// TIA Portal V15.1 export
// export: Created 2024-06-21T08:41:21.2804281Z, ExportSetting WithDefaults, DisplayName Totally Integrated Automation Portal, DisplayVersion V15.1 Update 5, DisplayName TIA Portal Openness, DisplayVersion V15.1 Update 5, DisplayName SINAMICS Startdrive Advanced, DisplayVersion V15.1, DisplayName G130, G150, S120, S150, SINAMICS MV, S210, DisplayVersion V15.1, DisplayName G110M, G120, G120C, G120D, G120P, DisplayVersion V15.1, DisplayName STEP 7 Professional, DisplayVersion V15.1 Update 5, DisplayName STEP 7 Safety, DisplayVersion V15.1, DisplayName WinCC Professional, DisplayVersion V15.1 Update 5, DisplayName SIMATIC Visualization Architect, DisplayVersion V15.1
FUNCTION_BLOCK "LVIDSDeCouple"   // FB1208, SCL
{ S7_Optimized_Access := 'TRUE' }
VERSION : 0.1
// stored: AutoNumber false, IsIECCheckEnabled false, IsRetainMemResEnabled false, MemoryReserve 100, SetENOAutomatically False, UDAEnableTagReadback false
   VAR_INPUT
      C_SoftCouple { ExternalAccessible := 'False'; ExternalVisible := 'False'; ExternalWritable := 'False'} : Bool;   // If true, coupling between CarrierID and BodyID or Mixnumber, otherwise with TagID
      I_DataModeManEn { ExternalAccessible := 'False'; ExternalVisible := 'False'; ExternalWritable := 'False'} : Bool;   // Dat mode manual enabled
      I_TagID { ExternalAccessible := 'False'; ExternalVisible := 'False'; ExternalWritable := 'False'} : DWord;   // Received TagId to couple with Data / Tag ID (0 if not used)
      I_BodyID { ExternalAccessible := 'False'; ExternalVisible := 'False'; ExternalWritable := 'False'} : DWord;   // Bodynumber (0 if not used)
      I_CarrierID { ExternalAccessible := 'False'; ExternalVisible := 'False'; ExternalWritable := 'False'} : DWord;   // Carrier ID
      I_MixNbr { ExternalAccessible := 'False'; ExternalVisible := 'False'; ExternalWritable := 'False'} : DWord;   // Mixnumber (0 if not used)
      I_PopID { ExternalAccessible := 'False'; ExternalVisible := 'False'; ExternalWritable := 'False'} : UDInt;   // Spare Data / PopID (0 if not used)
      I_PopIDSuffix { ExternalAccessible := 'False'; ExternalVisible := 'False'; ExternalWritable := 'False'} : Char;   // PopID suffix (' ' if not used)
      I_PopType { ExternalAccessible := 'False'; ExternalVisible := 'False'; ExternalWritable := 'False'} : UDInt;   // Pop identifier
      I_Start { ExternalAccessible := 'False'; ExternalVisible := 'False'; ExternalWritable := 'False'} : Bool;   // Start command for coupling / Start command
   END_VAR
   VAR_OUTPUT
      O_DataModeAuto { ExternalAccessible := 'False'; ExternalVisible := 'False'; ExternalWritable := 'False'} : Bool;   // Couple or decouple in automatic mode / Data mode - Automatic
      O_DataModeMan { ExternalAccessible := 'False'; ExternalVisible := 'False'; ExternalWritable := 'False'} : Bool;   // Data mode - Manual
      O_Busy { ExternalAccessible := 'False'; ExternalVisible := 'False'; ExternalWritable := 'False'} : Bool;   // Coupling busy
      O_Status { ExternalAccessible := 'False'; ExternalVisible := 'False'; ExternalWritable := 'False'} : Int;   // Status / Status (< 0 : alarm)
      O_Alarm { ExternalAccessible := 'False'; ExternalVisible := 'False'; ExternalWritable := 'False'} : Bool;   // Alarm
      O_OK { ExternalAccessible := 'False'; ExternalVisible := 'False'; ExternalWritable := 'False'} : Bool;   // Coupling or decoupling done OK / Coupling OK
      O_NOK { ExternalAccessible := 'False'; ExternalVisible := 'False'; ExternalWritable := 'False'} : Bool;   // Coupling or decoupling done NOK / Coupling NOK
   END_VAR
   VAR_IN_OUT
      IO_VIDS : "VIDS";   // VIDS internal record
      IO_VEMData : "VEMData";   // VEM data (From master)
      IO_Alarm : "Alarm";   // Alarm
      H_DeCouple : "H_LVIDSDeCouple";
      H_HMI : "H_HMI";
   END_VAR
   VAR
      DataModeAuto { ExternalAccessible := 'False'; ExternalVisible := 'False'; ExternalWritable := 'False'} : Bool;   // Couple or decouple in automode
      DataModeAutoPls { ExternalAccessible := 'False'; ExternalVisible := 'False'; ExternalWritable := 'False'} : Bool;
      DataModeMan { ExternalAccessible := 'False'; ExternalVisible := 'False'; ExternalWritable := 'False'} : Bool;
      DataModeManPls { ExternalAccessible := 'False'; ExternalVisible := 'False'; ExternalWritable := 'False'} : Bool;
      DataModeEdit { ExternalAccessible := 'False'; ExternalVisible := 'False'; ExternalWritable := 'False'} : Bool;
      DataModeMem { ExternalAccessible := 'False'; ExternalVisible := 'False'; ExternalWritable := 'False'} : Int;
      DataModeChanged { ExternalAccessible := 'False'; ExternalVisible := 'False'; ExternalWritable := 'False'} : Bool;
      DeCoupleBeginReqPlsAuto { ExternalAccessible := 'False'; ExternalVisible := 'False'; ExternalWritable := 'False'} : Bool;
      DeCoupleBeginReqPlsMan { ExternalAccessible := 'False'; ExternalVisible := 'False'; ExternalWritable := 'False'} : Bool;
      StartPls { ExternalAccessible := 'False'; ExternalVisible := 'False'; ExternalWritable := 'False'} : Bool;
      BeginReqAuto { ExternalAccessible := 'False'; ExternalVisible := 'False'; ExternalWritable := 'False'} : Bool;
      Busy { ExternalAccessible := 'False'; ExternalVisible := 'False'; ExternalWritable := 'False'} : Bool;
      BeginReqMan { ExternalAccessible := 'False'; ExternalVisible := 'False'; ExternalWritable := 'False'} : Bool;
      CarrierID { ExternalAccessible := 'False'; ExternalVisible := 'False'; ExternalWritable := 'False'} : DWord;
      CarrierIDValid { ExternalAccessible := 'False'; ExternalVisible := 'False'; ExternalWritable := 'False'} : Bool;
   END_VAR
   VAR DB_SPECIFIC
      CarrierIDMem { ExternalAccessible := 'False'; ExternalVisible := 'False'; ExternalWritable := 'False'} : DWord;   // Memory of CarrierID at begin request
   END_VAR
   VAR
      Identification { ExternalAccessible := 'False'; ExternalVisible := 'False'; ExternalWritable := 'False'} : DWord;
      IdentificationValid { ExternalAccessible := 'False'; ExternalVisible := 'False'; ExternalWritable := 'False'} : Bool;
      IdentificationMem { ExternalAccessible := 'False'; ExternalVisible := 'False'; ExternalWritable := 'False'} : DWord;
      BodyNbr { ExternalAccessible := 'False'; ExternalVisible := 'False'; ExternalWritable := 'False'} : DWord;
      BodyNbrValid { ExternalAccessible := 'False'; ExternalVisible := 'False'; ExternalWritable := 'False'} : Bool;
      BodyIDMem { ExternalAccessible := 'False'; ExternalVisible := 'False'; ExternalWritable := 'False'} : DWord;
      MixNbr { ExternalAccessible := 'False'; ExternalVisible := 'False'; ExternalWritable := 'False'} : DWord;
      MixNbrValid { ExternalAccessible := 'False'; ExternalVisible := 'False'; ExternalWritable := 'False'} : Bool;
      MixNbrMem { ExternalAccessible := 'False'; ExternalVisible := 'False'; ExternalWritable := 'False'} : DWord;
      PopIDMem { ExternalAccessible := 'False'; ExternalVisible := 'False'; ExternalWritable := 'False'} : DWord;
      PopIDSuffixMem { ExternalAccessible := 'False'; ExternalVisible := 'False'; ExternalWritable := 'False'} : Char;
      PopTypeMem { ExternalAccessible := 'False'; ExternalVisible := 'False'; ExternalWritable := 'False'} : DWord;
      DataValid { ExternalAccessible := 'False'; ExternalVisible := 'False'; ExternalWritable := 'False'} : Bool;
      InputDataValidAuto { ExternalAccessible := 'False'; ExternalVisible := 'False'; ExternalWritable := 'False'} : Bool;
      InputDataValidMan { ExternalAccessible := 'False'; ExternalVisible := 'False'; ExternalWritable := 'False'} : Bool;
      DataNotValid { ExternalAccessible := 'False'; ExternalVisible := 'False'; ExternalWritable := 'False'} : Bool;
   END_VAR
   VAR DB_SPECIFIC
      BeginPlsModeAuto { ExternalAccessible := 'False'; ExternalVisible := 'False'; ExternalWritable := 'False'} : Bool;   // Pulse of begin in auto mode
      BeginPlsModeManTagId { ExternalAccessible := 'False'; ExternalVisible := 'False'; ExternalWritable := 'False'} : Bool;   // Pulse of begin in manual mode
      BeginReqPls { ExternalAccessible := 'False'; ExternalVisible := 'False'; ExternalWritable := 'False'} : Bool;   // Pulse of begin request
      TagIdModeManMem { ExternalAccessible := 'False'; ExternalVisible := 'False'; ExternalWritable := 'False'} : DWord;   // Memorised TagId in manual mode
      Alarm { ExternalAccessible := 'False'; ExternalVisible := 'False'; ExternalWritable := 'False'} : Bool;   // Alarm
      ChangedRcvDataAlarm { ExternalAccessible := 'False'; ExternalVisible := 'False'; ExternalWritable := 'False'} : Bool;   // Alarm received data has chnged after request
      CoupleAlarm { ExternalAccessible := 'False'; ExternalVisible := 'False'; ExternalWritable := 'False'} : Bool;   // Alarm couple or decouple NOK
      Status { ExternalAccessible := 'False'; ExternalVisible := 'False'; ExternalWritable := 'False'} : Int;   // Status
   END_VAR
   VAR
      btnDataModeAutoColour { ExternalAccessible := 'False'; ExternalVisible := 'False'; ExternalWritable := 'False'} : Word;
      btnDataModeManColour { ExternalAccessible := 'False'; ExternalVisible := 'False'; ExternalWritable := 'False'} : Word;
      btnDeCoupleVisible { ExternalAccessible := 'False'; ExternalVisible := 'False'; ExternalWritable := 'False'} : Word;
      btnDeCoupleEnable { ExternalAccessible := 'False'; ExternalVisible := 'False'; ExternalWritable := 'False'} : Word;
      btnDeCouplePls { ExternalAccessible := 'False'; ExternalVisible := 'False'; ExternalWritable := 'False'} : Bool;
      btnEditVisible { ExternalAccessible := 'False'; ExternalVisible := 'False'; ExternalWritable := 'False'} : Word;
      btnEditEnable { ExternalAccessible := 'False'; ExternalVisible := 'False'; ExternalWritable := 'False'} : Word;
      msgVEMDataBodyVisible { ExternalAccessible := 'False'; ExternalVisible := 'False'; ExternalWritable := 'False'} : Word;
      msgVEMDataCarrierVisible { ExternalAccessible := 'False'; ExternalVisible := 'False'; ExternalWritable := 'False'} : Word;
      msgDataValidVisible { ExternalAccessible := 'False'; ExternalVisible := 'False'; ExternalWritable := 'False'} : Word;   // HMI - Couple/Decouple OK
      msgDataNotValidVisible { ExternalAccessible := 'False'; ExternalVisible := 'False'; ExternalWritable := 'False'} : Word;   // HMI - Couple/Decouple OK
      msgPartPresVisible { ExternalAccessible := 'False'; ExternalVisible := 'False'; ExternalWritable := 'False'} : Word;
      txtCarrierIDDeCoupleVisible { ExternalAccessible := 'False'; ExternalVisible := 'False'; ExternalWritable := 'False'} : Word;
      txtCarrierIDDeCoupleEnable { ExternalAccessible := 'False'; ExternalVisible := 'False'; ExternalWritable := 'False'} : Word;
      txtCarrierIDDeCoupleColour { ExternalAccessible := 'False'; ExternalVisible := 'False'; ExternalWritable := 'False'} : Word;
      txtCarrierIDDeCoupleValid { ExternalAccessible := 'False'; ExternalVisible := 'False'; ExternalWritable := 'False'} : Bool;
      txtIdentificationDeCoupleVisible { ExternalAccessible := 'False'; ExternalVisible := 'False'; ExternalWritable := 'False'} : Word;
      txtIdentificationDeCoupleEnable { ExternalAccessible := 'False'; ExternalVisible := 'False'; ExternalWritable := 'False'} : Word;
      txtIdentificationDeCoupleColour { ExternalAccessible := 'False'; ExternalVisible := 'False'; ExternalWritable := 'False'} : Word;
      txtIdentificationDeCoupleValid { ExternalAccessible := 'False'; ExternalVisible := 'False'; ExternalWritable := 'False'} : Bool;
      txtMixNbrDeCoupleVisible { ExternalAccessible := 'False'; ExternalVisible := 'False'; ExternalWritable := 'False'} : Word;
      txtMixNbrDeCoupleEnable { ExternalAccessible := 'False'; ExternalVisible := 'False'; ExternalWritable := 'False'} : Word;
      txtMixNbrDeCoupleColour { ExternalAccessible := 'False'; ExternalVisible := 'False'; ExternalWritable := 'False'} : Word;
      txtMixNbrDeCoupleValid { ExternalAccessible := 'False'; ExternalVisible := 'False'; ExternalWritable := 'False'} : Bool;
      txtBodyIDDeCoupleVisible { ExternalAccessible := 'False'; ExternalVisible := 'False'; ExternalWritable := 'False'} : Word;
      txtBodyIDDeCoupleEnable { ExternalAccessible := 'False'; ExternalVisible := 'False'; ExternalWritable := 'False'} : Word;
      txtBodyIDDeCoupleColour { ExternalAccessible := 'False'; ExternalVisible := 'False'; ExternalWritable := 'False'} : Word;
      txtBodyIDDeCoupleValid { ExternalAccessible := 'False'; ExternalVisible := 'False'; ExternalWritable := 'False'} : Bool;
      txtPopIDDeCoupleVisible { ExternalAccessible := 'False'; ExternalVisible := 'False'; ExternalWritable := 'False'} : Word;
      txtPopIDDeCoupleEnable { ExternalAccessible := 'False'; ExternalVisible := 'False'; ExternalWritable := 'False'} : Word;
      txtPopIDDeCoupleColour { ExternalAccessible := 'False'; ExternalVisible := 'False'; ExternalWritable := 'False'} : Word;
      txtPopIDDeCoupleValid { ExternalAccessible := 'False'; ExternalVisible := 'False'; ExternalWritable := 'False'} : Bool;
      txtPopIDSuffixDeCoupleVisible { ExternalAccessible := 'False'; ExternalVisible := 'False'; ExternalWritable := 'False'} : Word;
      txtPopIDSuffixDeCoupleEnable { ExternalAccessible := 'False'; ExternalVisible := 'False'; ExternalWritable := 'False'} : Word;
      txtPopIDSuffixDeCoupleColour { ExternalAccessible := 'False'; ExternalVisible := 'False'; ExternalWritable := 'False'} : Word;
      txtPopTypeDeCoupleVisible { ExternalAccessible := 'False'; ExternalVisible := 'False'; ExternalWritable := 'False'} : Word;
      txtPopTypeDeCoupleEnable { ExternalAccessible := 'False'; ExternalVisible := 'False'; ExternalWritable := 'False'} : Word;
      txtPopTypeDeCoupleColour { ExternalAccessible := 'False'; ExternalVisible := 'False'; ExternalWritable := 'False'} : Word;
      IconColour { ExternalAccessible := 'False'; ExternalVisible := 'False'; ExternalWritable := 'False'} : Word;
      DeCoupleOK { ExternalAccessible := 'False'; ExternalVisible := 'False'; ExternalWritable := 'False'} : Bool;
      DeCoupleNOK { ExternalAccessible := 'False'; ExternalVisible := 'False'; ExternalWritable := 'False'} : Bool;
      _DataModeManForcedPls { ExternalAccessible := 'False'; ExternalVisible := 'False'; ExternalWritable := 'False'; S7_SetPoint := 'True'} : R_TRIG;
      _DataModeAutoPls { ExternalAccessible := 'False'; ExternalVisible := 'False'; ExternalWritable := 'False'; S7_SetPoint := 'True'} : R_TRIG;
      _DeCoupleStartPls { ExternalAccessible := 'False'; ExternalVisible := 'False'; ExternalWritable := 'False'; S7_SetPoint := 'True'} : R_TRIG;
      _DataModeChangedPls { ExternalAccessible := 'False'; ExternalVisible := 'False'; ExternalWritable := 'False'; S7_SetPoint := 'True'} : R_TRIG;
      _btnDeCouplePls { ExternalAccessible := 'False'; ExternalVisible := 'False'; ExternalWritable := 'False'; S7_SetPoint := 'True'} : R_TRIG;
   END_VAR
   VAR CONSTANT
      STATUS_OK : Int := 1;
      STATUS_COUPLE_REQ : Int := 107;
      STATUS_COUPLE_RUNNING : Int := 207;
      STATUS_DECOUPLE_REQ : Int := 108;
      STATUS_DECOUPLE_RUNNING : Int := 208;
      OFF : Word := 2#0000000000000000;
      ON : Word := 2#0000000000000001;
      VISIBLE : Word := 2#0000000000000001;
      ENABLE : Word := 2#0000000000000010;
      BG_COLOUR_GREY : Word := 2#0000000000000100;
      COLOUR_DEFAULT : Word := 2#0000000000000000;
      COLOUR_RED : Word := 2#0000000000010000;
      COLOUR_GREEN : Word := 2#0000000000100000;
      COLOUR_BLUE : Word := 2#0000000001000000;
      COLOUR_WHITE : Word := 2#0000000010000000;
      BG_COLOUR_BLUE_FLASH : Word := 2#0000000010000000;
      BG_COLOUR_LIGHTRED : Word := 2#0100000000000000;
      BG_COLOUR_YELLOW : Word := 2#1000000000000000;
      OK_BEGIN_DELAY_MAX : Time := T#10s;
      CMD_DECOUPLE : DWord := 2006;
   END_VAR
BEGIN
   (******************************************************************************)
   (* Data mode - Activation                                                     *)
   (******************************************************************************)

   //Automatic
   //Data mode selected  - No mode, select auto
   IF (#H_DeCouple.H_selDataMode < 1) OR (#H_DeCouple.H_selDataMode > 3) OR NOT #IO_VIDS.PartPres OR NOT #I_DataModeManEn THEN
       #H_DeCouple.H_selDataMode := 1;
   END_IF;

   //Data mode automatic - Activation
   #DataModeAuto := (#H_DeCouple.H_selDataMode = 1);

   //Data mode automatic - Create pulse upon selection 
   #_DataModeAutoPls(CLK:=#DataModeAuto,Q=>#DataModeAutoPls);

   //Data mode manual - Activation
   #DataModeMan := (#H_DeCouple.H_selDataMode = 2);

   //Data mode manual - Create pulse upon selection
   #_DataModeManForcedPls(CLK := #DataModeMan,Q => #DataModeManPls);

   //Data mode changed
   #_DataModeAutoPls(CLK := #H_DeCouple.H_selDataMode <> #DataModeMem,Q => #DataModeAutoPls);
   #DataModeMem:=#H_DeCouple.H_selDataMode;

   //Data mode edit - Activation
   IF #DataModeMan AND (#H_DeCouple.H_btnEdit = #ON) THEN
       #DataModeEdit := TRUE;
       //Copy VEM data to HMI
       #H_DeCouple.H_txtIdentification := #IO_VEMData.Identification;

   ELSIF #DataModeAuto THEN
       #DataModeEdit := FALSE;
   END_IF;


   IF #DataModeEdit THEN

       //Check valid
       #txtCarrierIDDeCoupleValid := #H_DeCouple.H_txtCarrierIDDeCouple > 0;
       #txtIdentificationDeCoupleValid := #H_DeCouple.H_txtIdentificationDeCouple > 0;
       #txtBodyIDDeCoupleValid :=#H_DeCouple.H_txtBodyIDDeCouple > 0;
       #txtMixNbrDeCoupleValid := #H_DeCouple.H_txtMixNbrDeCouple > 0;
       #txtPopIDDeCoupleValid := #H_DeCouple.H_txtPopIdDeCouple > 0;

       //Entry fields valid
       #InputDataValidMan := #txtCarrierIDDeCoupleValid AND (#txtIdentificationDeCoupleValid OR #txtBodyIDDeCoupleValid OR #txtMixNbrDeCoupleValid OR #txtPopIDDeCoupleValid);

   ELSE

       //Reset
       #InputDataValidMan := FALSE;

   END_IF;

   (******************************************************************************)
   (* Data mode automatic - Begin request                                        *)
   (******************************************************************************)

   //Start - Create pulse
   #_DeCoupleStartPls(CLK := #I_Start,
                    Q => #StartPls);

   #BeginReqAuto:=False;
   IF #DataModeAuto AND #StartPls AND #IO_VIDS.PartPres AND #I_CarrierID > 0  THEN

       //Memorize parameters
       #IdentificationMem := #I_TagID;
       #BodyIDMem := #I_BodyID;
       #CarrierIDMem := #I_CarrierID;
       #MixNbrMem := #I_MixNbr;
       #PopIDMem := #I_PopID;
       #PopIDSuffixMem := #I_PopIDSuffix;
       #PopTypeMem := #I_PopType;

       //Data mode automatic - Begin request
       #BeginReqAuto := True;

   END_IF;

   (******************************************************************************)
   (* Data mode manual - Begin request                                           *)
   (******************************************************************************)

   //Couple button - Create pulse 
   #_btnDeCouplePls(CLK:=#H_DeCouple.H_btnDecouple=#ON,
                  Q=>#btnDeCouplePls);

   #BeginReqMan := False;
   IF #DataModeEdit AND #btnDeCouplePls AND #IO_VIDS.PartPres THEN

       //Edit mode off
       #DataModeEdit := FALSE;

       //Memorize data
       #CarrierIDMem := #H_DeCouple.H_txtCarrierIDDeCouple;

       //Start with a clean sheet
       #IdentificationMem := 0;
       #BodyIDMem := 0;
       #MixNbrMem := 0;
       #PopIDMem := 0;
       #PopIDSuffixMem := ' ';
       #PopTypeMem := 0;

       //Memorize parameters
       IF #H_DeCouple.H_txtIdentificationDeCouple > 0 THEN
           #IdentificationMem := #H_DeCouple.H_txtIdentificationDeCouple;
       ELSIF #H_DeCouple.H_txtBodyIDDeCouple > 0 THEN
           #BodyIDMem := #H_DeCouple.H_txtBodyIDDeCouple;
       ELSIF #H_DeCouple.H_txtMixNbrDeCouple > 0 THEN
           #MixNbrMem := #H_DeCouple.H_txtMixNbrDeCouple;
       ELSIF #H_DeCouple.H_txtPopIdDeCouple > 0 OR #H_DeCouple.H_txtPopIdSuffixDeCouple <> ' ' OR #H_DeCouple.H_txtPopTypeDeCouple <> 0  THEN
           #PopIDMem := #H_DeCouple.H_txtPopIdDeCouple;
           #PopIDSuffixMem := #H_DeCouple.H_txtPopIdSuffixDeCouple;
           #PopTypeMem := #H_DeCouple.H_txtPopTypeDeCouple;
       END_IF;

       //Data mode manual - begin request
       #BeginReqMan := True;

   END_IF;

   (******************************************************************************)
   (* Begin request - Summary                                                    *)
   (******************************************************************************)

   #IO_VIDS.DeCouple.BeginReq := #BeginReqAuto OR #BeginReqMan;

   IF #IO_VIDS.DeCouple.BeginReq THEN
       #DeCoupleOK := False;
       #DeCoupleNOK := False;
   END_IF;

   (*******************************************************)
   (* Begin                                               *)
   (*******************************************************)

   IF #IO_VIDS.DeCouple.OkBegin THEN
       //Initialize parameters
       #IO_VIDS.VEMData.IdType := #IO_VIDS.IDType;
       #IO_VIDS.VEMData.FunctionCode := 255;
       #IO_VIDS.VEMData.Identification := #IdentificationMem;
       #IO_VIDS.VEMData.BodyID := #BodyIDMem;
       #IO_VIDS.VEMData.CarrierID := #CarrierIDMem;
       #IO_VIDS.VEMData.MixNumber := #MixNbrMem;
       #IO_VIDS.VEMData.PopID := #PopIDMem;
       #IO_VIDS.VEMData.PopIDSuffix := #PopIDSuffixMem;
       #IO_VIDS.VEMData.PopType := #PopTypeMem;
       #IO_VIDS.VEMData.CommandCode := #CMD_DECOUPLE;
       #Status := #IO_VIDS.DeCouple.Status;
   END_IF;

   #IO_VIDS.DeCouple.Begin := #IO_VIDS.DeCouple.OkBegin;

   (*******************************************************)
   (* Running                                             *)
   (*******************************************************)
   IF #IO_VIDS.DeCouple.Running THEN
       #Status := #IO_VIDS.DeCouple.Status;
   END_IF;

   #Busy := #IO_VIDS.DeCouple.Running;

   (*******************************************************)
   (* Finish                                              *)
   (*******************************************************)

   IF #IO_VIDS.DeCouple.Finished THEN

       //Update status
       #Status := #IO_VIDS.DeCouple.Status;

       //Status OK/NOK
       IF #Status = #STATUS_OK THEN
           #DeCoupleOK := True;
       ELSE
           #DeCoupleNOK := True;
           IF #DataModeMan THEN
               #DataModeEdit := TRUE;
           END_IF;
       END_IF;

   END_IF;

   (******************************************************************************)
   (* Alarm                                                                      *)
   (******************************************************************************)

   #Alarm := (#Status < 0);

   "LAlarmSummary"(I_AlarmA := "FALSE",
                   I_AlarmB := "FALSE",
                   I_AlarmC := #Alarm,
                   I_AlarmD := "FALSE",
                   I_AlarmABCondition := "FALSE",
                   IO_Alarm := #IO_Alarm,
                   C_UpperLevelHW := "FALSE",
                   C_UpperLevelSafety := "FALSE",
                   C_Safety := "FALSE",
                   C_Mechanic := "FALSE",
                   C_Transport := "FALSE",
                   C_Feature1 := "FALSE",
                   C_Feature2 := "FALSE",
                   C_Feature3 := "FALSE");


   (*******************************************************)
   (* Reset                                               *)
   (*******************************************************)

   IF NOT #IO_VIDS.PartPres THEN
       #DeCoupleOK := False;
       #DeCoupleNOK := False;
       #H_DeCouple.H_txtIdentification := 0;
       #H_DeCouple.H_txtBodyID := 0;
       #H_DeCouple.H_txtCarrierID := 0;
       #H_DeCouple.H_txtMixNbr := 0;
       #H_DeCouple.H_txtPopId := 0;
       #H_DeCouple.H_txtPopIdSuffix := ' ';
       #H_DeCouple.H_txtPopType := 0;
       #Status := 0;
   END_IF;

   (*******************************************************)
   (* Outputs                                             *)
   (*******************************************************)

   #O_DataModeAuto := #DataModeAuto;
   #O_DataModeMan := #DataModeMan;
   #O_OK := #DeCoupleOK;
   #O_NOK := #DeCoupleNOK;

   #O_Busy := #Busy;
   #O_Status := #Status;
   #O_Alarm := #Status < 0;

   (*******************************************************)
   (* HMI - Reset buttons                                 *)
   (*******************************************************)

   #H_DeCouple.H_btnEdit := #OFF;
   #H_DeCouple.H_btnDecouple := #OFF;
   #H_DeCouple.H_btnDecouple := #OFF;

   (*******************************************************)
   (* HMI - Update text fields                            *)
   (*******************************************************)

   IF #IO_VIDS.VEMDataValid THEN
       #H_DeCouple.H_txtCarrierIDDeCouple := #IO_VEMData.CarrierID;
       #H_DeCouple.H_txtIdentificationDeCouple := #IO_VEMData.Identification;
       #H_DeCouple.H_txtBodyIDDeCouple := #IO_VEMData.BodyID;
       #H_DeCouple.H_txtMixNbrDeCouple := #IO_VEMData.MixNumber;
       #H_DeCouple.H_txtPopId := #IO_VEMData.PopID;
       #H_DeCouple.H_txtPopIdSuffix := #IO_VEMData.PopIDSuffix;
       #H_DeCouple.H_txtPopType := #IO_VEMData.PopType;
   ELSE
       #H_DeCouple.H_txtCarrierID := 0;
       #H_DeCouple.H_txtIdentification := 0;
       #H_DeCouple.H_txtBodyID := 0;
       #H_DeCouple.H_txtMixNbr := 0;
       #H_DeCouple.H_txtPopId := 0;
       #H_DeCouple.H_txtPopIdSuffix := ' ';
       #H_DeCouple.H_txtPopType := 0;
   END_IF;

   (*******************************************************)
   (* HMI - Input fields                                  *)
   (*******************************************************)

   //Visible
   #txtIdentificationDeCoupleVisible := #OFF;
   #txtBodyIDDeCoupleVisible := #OFF;
   #txtCarrierIDDeCoupleVisible := #OFF;
   #txtMixNbrDeCoupleVisible := #OFF;
   #txtPopIDDeCoupleVisible := #OFF;
   #txtPopIDSuffixDeCoupleVisible := #OFF;
   #txtPopTypeDeCoupleVisible := #OFF;

   IF #DataModeMan THEN
       #txtCarrierIDDeCoupleVisible := #VISIBLE;
       IF #C_SoftCouple THEN
           #txtBodyIDDeCoupleVisible := #VISIBLE;
           #txtMixNbrDeCoupleVisible := #VISIBLE;
           #txtPopIDDeCoupleVisible := #VISIBLE;
           #txtPopIDSuffixDeCoupleVisible := #VISIBLE;
           #txtPopTypeDeCoupleVisible := #VISIBLE;
       ELSE
           #txtIdentificationDeCoupleVisible := #VISIBLE;
       END_IF;
   END_IF;

   //Enable
   #txtIdentificationDeCoupleEnable := #OFF;
   #txtCarrierIDDeCoupleEnable := #OFF;
   #txtBodyIDDeCoupleEnable := #OFF;
   #txtMixNbrDeCoupleEnable := #OFF;
   #txtPopIDDeCoupleEnable := #OFF;
   #txtPopIDSuffixDeCoupleEnable := #OFF;
   #txtPopTypeDeCoupleEnable := #OFF;

   IF #DataModeEdit THEN
       #txtCarrierIDDeCoupleEnable := #ENABLE;
       IF #C_SoftCouple THEN
           #txtBodyIDDeCoupleEnable := #ENABLE;
           #txtMixNbrDeCoupleEnable := #ENABLE;
           #txtPopIDDeCoupleEnable := #ENABLE;
           #txtPopIDSuffixDeCoupleEnable := #ENABLE;
           #txtPopTypeDeCoupleEnable := #ENABLE;
       ELSE
           #txtIdentificationDeCoupleEnable := #ENABLE;
       END_IF;
   END_IF;

   (*******************************************************)
   (* HMI - Buttons                                       *)
   (*******************************************************)

   //HMI - Button Data mode automatic
   IF #DataModeAuto THEN
       #btnDataModeAutoColour := #COLOUR_GREEN;
   ELSE
       #btnDataModeAutoColour := #COLOUR_DEFAULT;
   END_IF;

   //HMI - Button Data mode manual
   IF #DataModeMan THEN
       #btnDataModeManColour := #COLOUR_BLUE;
   ELSE
       #btnDataModeManColour := #COLOUR_DEFAULT;
   END_IF;

   //HMI - Button Edit
   IF #DataModeMan AND NOT #DataModeEdit AND NOT #IO_VIDS.Couple.Running THEN
       #btnEditVisible := #VISIBLE;
       #btnEditEnable := #ENABLE;
   ELSE
       #btnEditVisible := #OFF;
       #btnEditEnable := #OFF;
   END_IF;

   //HMI - Button Couple
   IF #DataModeEdit AND #InputDataValidMan THEN
       #btnDeCoupleVisible := #VISIBLE;
       #btnDeCoupleEnable := #ENABLE;
   ELSE
       #btnDeCoupleVisible := #OFF;
       #btnDeCoupleEnable := #OFF;
   END_IF;

   (*******************************************************)
   (* HMI - Messages                                      *)
   (*******************************************************)

   //HMI - Message part present
   IF #IO_VIDS.PartPres THEN
       #msgPartPresVisible := #VISIBLE;
   ELSE
       #msgPartPresVisible := #OFF;
   END_IF;

   //HMI - Message data valid, not valid
   IF #IO_VIDS.VEMDataValid THEN
       #msgDataValidVisible := #VISIBLE;
   ELSIF #IO_VIDS.VEMDataNotValid THEN
       #msgDataNotValidVisible := #VISIBLE;
   ELSE
       #msgDataValidVisible := #OFF;
       #msgDataNotValidVisible := #OFF;
   END_IF;

   //Body or carrier data
   IF #IO_VIDS.IDType = 0 THEN
       #msgVEMDataBodyVisible := #VISIBLE;
       #msgVEMDataCarrierVisible := #OFF;
   ELSE
       #msgVEMDataBodyVisible := #OFF;
       #msgVEMDataCarrierVisible := #VISIBLE;
   END_IF;

   (*******************************************************)
   (* Icon - animation                                    *)
   (*******************************************************)

   "LIAnimDWord"(I_SetPos:=FALSE,
                   I_ResetPos:=FALSE,
                   I_Active:=#Status>1,
                   I_Visible:=FALSE,
                   I_OutOfUse:=FALSE,
                   I_IntlkSet:=FALSE,
                   I_IntlkReset:=FALSE,
                   I_IntlkSetAlm:=FALSE,
                   I_IntlkResetAlm:=FALSE,
                   I_ManualMode:=#DataModeMan,
                   I_FncSelInHMI:=FALSE,
                   I_AnySelected:=FALSE,
                   I_AlarmA:=FALSE,
                   I_AlarmB:=FALSE,
                   I_AlarmC:=#Status<0,
                   I_AlarmD:=FALSE,
                   I_SafetyOk:=FALSE,
                   I_Service:="TRUE",
                 I_Spare1:="FALSE",
                 I_Spare2:="FALSE",
                 I_Spare3:="FALSE",
                 I_Spare4:="FALSE",
                 I_Spare5:="FALSE",
                 I_Spare6:="FALSE",
                 I_Spare7:="FALSE",
                 I_Spare8:="FALSE",
                 I_Spare9:="FALSE",
                 I_Spare10:="FALSE",
                 I_Spare11:="FALSE",
                 I_Spare12:="FALSE",
                 I_Spare13:="FALSE",
                 I_Spare14:="FALSE",
                 H_IAnim=>#H_HMI.H_IAnim);

   (*******************************************************)
   (* HMI - Animations summary                            *)
   (*******************************************************)

   #H_DeCouple.H_txtCommandCodeSent := #IO_VIDS.CmdCodeSent;
   #H_DeCouple.H_txtCommandCodeRcvd := #IO_VIDS.CmdCodeRcvd;
   #H_DeCouple.H_msgVEMDataBodyAnim := #msgVEMDataBodyVisible;
   #H_DeCouple.H_msgVEMDataCarrierAnim := #msgVEMDataCarrierVisible;
   #H_DeCouple.H_btnDataModeAutoAnim := #btnDataModeAutoColour;
   #H_DeCouple.H_btnDataModeManAnim := #btnDataModeManColour;
   #H_DeCouple.H_txtCarrierIDDeCoupleAnim := #txtCarrierIDDeCoupleVisible OR #txtCarrierIDDeCoupleEnable OR #txtCarrierIDDeCoupleColour;
   #H_DeCouple.H_txtIdentificationDeCoupleAnim := #txtIdentificationDeCoupleVisible OR #txtIdentificationDeCoupleEnable OR #txtIdentificationDeCoupleColour;
   #H_DeCouple.H_txtBodyIDDeCoupleAnim := #txtBodyIDDeCoupleVisible OR #txtBodyIDDeCoupleEnable OR #txtBodyIDDeCoupleColour;
   #H_DeCouple.H_txtMixNbrDeCoupleAnim := #txtMixNbrDeCoupleVisible OR #txtMixNbrDeCoupleEnable OR #txtMixNbrDeCoupleColour;
   #H_DeCouple.H_txtPopIdDeCoupleAnim := #txtPopIDDeCoupleVisible OR #txtPopIDDeCoupleEnable OR #txtPopIDDeCoupleColour;
   #H_DeCouple.H_txtPopIdSuffixDeCoupleAnim := #txtPopIDSuffixDeCoupleVisible OR #txtPopIDSuffixDeCoupleEnable OR #txtPopIDSuffixDeCoupleColour;
   #H_DeCouple.H_txtPopTypeDeCoupleAnim := #txtPopTypeDeCoupleVisible OR #txtPopTypeDeCoupleEnable OR #txtPopTypeDeCoupleColour;
   #H_DeCouple.H_btnEditAnim := #btnEditVisible OR #btnEditEnable;
   #H_DeCouple.H_btnDecoupleAnim := #btnDeCoupleVisible OR #btnDeCoupleEnable;
   #H_DeCouple.H_msgPartPresAnim := #msgPartPresVisible;
   #H_DeCouple.H_msgVEMDataValidAnim := #msgDataValidVisible;
   #H_DeCouple.H_msgVEMDataNotValidAnim := #msgDataNotValidVisible;
   #H_DeCouple.H_msgStatus := #Status;
END_FUNCTION_BLOCK
